Universal Robots PolyScope program: wrs2020_taskboard_pulley.urp

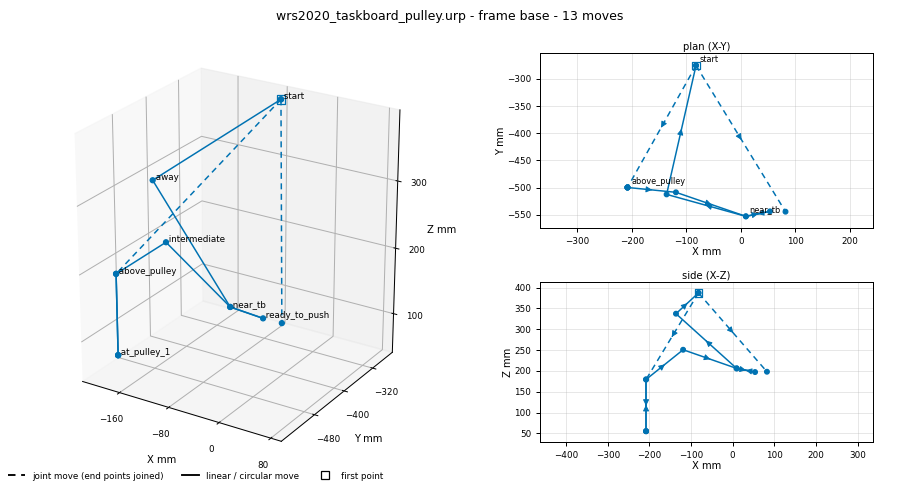
[picture p0: tool path of wrs2020_taskboard_pulley.urp in frame base, 13 of 13 moves have a stored position in this frame; points joined in program order, loops and branches not executed]
Program wrs2020_taskboard_pulley (installation=default directory=/programs/usbdisk createdIn=5.6.0.90886 lastSavedIn=5.6.0.90886 robotSerialNumber=20205500180)
Calibrated DH parameters: a=[0.000135, -0.030981, -0.334292, 0.000083, 0.000088, 0]; d=[0.162656, 258.79096, -331.603246, 72.945842, 0.099724, 0.099562]; alpha=[1.569535, 0.001639, 0.002824, 1.569633, -1.569323, 0]; deltaTheta=[0, 1.497881, -2.049261, 0.551379, 0, 0]
Robot Program (runOnlyOnce=true)
  MoveJ speed 60 deg/s, acceleration 80 deg/s^2 (useActiveTCP=false) tcp=gripper_140_tip; feature=Base
    Waypoint start: TCP in base x=-82.102 y=-275.549 z=387.348 mm, rx=-0.1814 ry=-3.1114 rz=0.2863 rad; joints [35.849, -127.007, 98.51, -68.6, -82.206, -47.132] deg; TCP offset x=0 y=0 z=220 mm, rx=0 ry=0 rz=0 rad
  URCap Gripper (Robotiq_Grippers, Robotiq Inc.) dataModel(position=44.705882352941174, force=100.0, speed=100.0, positionInDouble=44.705882352941174, forceInDouble=100.0, speedInDouble=100.0, slaveIds=[9], blocking=true)
  MoveJ speed 120 deg/s, acceleration 80 deg/s^2 (useActiveTCP=false) tcp=gripper_140_tip; feature=Base
    Waypoint above_pulley: TCP in base x=-208.011 y=-499.592 z=179.536 mm, rx=2.2188 ry=-2.2117 rz=-0.0634 rad; joints [54.601, -83.96, 96.653, -102.683, -92.188, -125.564] deg
  MoveL speed 250 mm/s, acceleration 1200 mm/s^2 (useActiveTCP=false) tcp=gripper_140_tip; feature=Base
    Waypoint at_pulley_1: motionParameters(jointSpeed=1.047198 jointAcceleration=1.396263 cartesianSpeed=0.5 cartesianAcceleration=1.2); TCP in base x=-208.011 y=-499.592 z=55.279 mm, rx=2.2188 ry=-2.2117 rz=-0.0634 rad; joints [54.587, -77.543, 108.66, -121.106, -92.18, -125.517] deg
  URCap Gripper (Robotiq_Grippers, Robotiq Inc.) dataModel(position=100.0, force=0.0, speed=0.0, positionInDouble=100.0, forceInDouble=0.0, speedInDouble=0.0, slaveIds=[9], blocking=true)
  URCap Gripper (Robotiq_Grippers, Robotiq Inc.) dataModel(position=56.86274509803921, force=0.0, speed=0.0, positionInDouble=56.86274509803921, forceInDouble=0.0, speedInDouble=0.0, slaveIds=[9], blocking=true)
  MoveL speed 500 mm/s, acceleration 1200 mm/s^2 (useActiveTCP=false) tcp=gripper_140_tip; feature=Base
    Waypoint at_pulley_2: motionParameters(jointSpeed=1.047198 jointAcceleration=1.396263 cartesianSpeed=0.5 cartesianAcceleration=1.2); TCP in base x=-207.996 y=-499.585 z=55.27 mm, rx=-0.009 ry=-3.1069 rz=-0.0353 rad; joints [54.588, -77.543, 108.661, -121.105, -92.181, -35] deg
  URCap Gripper (Robotiq_Grippers, Robotiq Inc.) dataModel(position=100.0, force=0.0, speed=0.0, positionInDouble=100.0, forceInDouble=0.0, speedInDouble=0.0, slaveIds=[9], blocking=true)
  URCap Gripper (Robotiq_Grippers, Robotiq Inc.) dataModel(position=56.86274509803921, force=0.0, speed=0.0, positionInDouble=56.86274509803921, forceInDouble=0.0, speedInDouble=0.0, slaveIds=[9], blocking=true)
  MoveL speed 500 mm/s, acceleration 1200 mm/s^2 (useActiveTCP=false) tcp=gripper_140_tip; feature=Base
    Waypoint at_pulley_1: motionParameters(jointSpeed=1.047198 jointAcceleration=1.396263 cartesianSpeed=0.5 cartesianAcceleration=1.2); TCP in base x=-208.011 y=-499.592 z=55.279 mm, rx=2.2188 ry=-2.2117 rz=-0.0634 rad; joints [54.587, -77.543, 108.66, -121.106, -92.18, -125.517] deg
  URCap Gripper (Robotiq_Grippers, Robotiq Inc.) dataModel(position=100.0, force=0.0, speed=0.0, positionInDouble=100.0, forceInDouble=0.0, speedInDouble=0.0, slaveIds=[9], blocking=true)
  MoveL speed 250 mm/s, acceleration 250 mm/s^2 (useActiveTCP=false) tcp=gripper_140_tip; feature=Base
    Waypoint above_pulley: TCP in base x=-208.011 y=-499.592 z=179.536 mm, rx=2.2188 ry=-2.2117 rz=-0.0634 rad; joints [54.601, -83.96, 96.653, -102.683, -92.188, -125.564] deg
    Waypoint intermediate: motionParameters(blendRadius=0.05); TCP in base x=-119.041 y=-508.485 z=250.905 mm, rx=-1.87 ry=2.1339 rz=-0.5992 rad; joints [46.177, -86.722, 91.166, -81.687, -65.2, -129.14] deg
  MoveL speed 250 mm/s, acceleration 250 mm/s^2 (useActiveTCP=false) tcp=gripper_140_tip; feature=Base
    Waypoint near_tb: TCP in base x=9.516 y=-552.663 z=206.118 mm, rx=-1.2151 ry=1.2878 rz=-1.2829 rad; joints [46.82, -54.652, 84.012, -32.299, -37.921, -179.667] deg
    Waypoint ready_to_push: TCP in base x=53.765 y=-543.482 z=197.335 mm, rx=-1.1908 ry=1.1936 rz=-1.2641 rad; joints [50.694, -52.534, 85.468, -29.603, -37.71, -184.158] deg
  Force Frame feature=Joint_6_name; selection=[1, 1, 1, 0, 0, 0]; wrench=[0, 0, 10, 0, 0, 0]; limitsForce=[0.15, 0.15, 0.01, 1.047198, 1.047198, 1.047198]; limitsMotion=[0.1, 0.1, 0.1, 0.349066, 0.349066, 0.349066]
    Wait Sleep waitTime=3
    Loop Counting (count=5) loopVariable(name=Loop_1)
      SuppressedNode
        MoveL speed 5 mm/s, acceleration 1200 mm/s^2 (useActiveTCP=true) feature=Base
          MoveDirectionNode (selectedDirection=XPlus toolParams=0.005, 1.2) feature=Joint_6_name
            Until DISTANCE (allowActions=false deceleration=3 distanceNodeType=STOP) Distance=0.002; motionParameters(blendRadius=0)
          MoveDirectionNode (selectedDirection=XMinus toolParams=0.005, 1.2) feature=Joint_6_name
            Until DISTANCE (allowActions=false deceleration=3 distanceNodeType=STOP) Distance=0.002; motionParameters(blendRadius=0)
          MoveDirectionNode (selectedDirection=XMinus toolParams=0.005, 1.2) feature=Joint_6_name
            Until DISTANCE (allowActions=false deceleration=3 distanceNodeType=STOP) Distance=0.002; motionParameters(blendRadius=0)
          MoveDirectionNode (selectedDirection=XPlus toolParams=0.005, 1.2) feature=Joint_6_name
            Until DISTANCE (allowActions=false deceleration=3 distanceNodeType=STOP) Distance=0.002; motionParameters(blendRadius=0)
          MoveDirectionNode (selectedDirection=YPlus toolParams=0.005, 1.2) feature=Joint_6_name
            Until DISTANCE (allowActions=false deceleration=3 distanceNodeType=STOP) Distance=0.002; motionParameters(blendRadius=0)
          MoveDirectionNode (selectedDirection=YMinus toolParams=0.005, 1.2) feature=Joint_6_name
            Until DISTANCE (allowActions=false deceleration=3 distanceNodeType=STOP) Distance=0.002; motionParameters(blendRadius=0)
          MoveDirectionNode (selectedDirection=YMinus toolParams=0.005, 1.2) feature=Joint_6_name
            Until DISTANCE (allowActions=false deceleration=3 distanceNodeType=STOP) Distance=0.002; motionParameters(blendRadius=0)
          MoveDirectionNode (selectedDirection=YPlus toolParams=0.005, 1.2) feature=Joint_6_name
            Until DISTANCE (allowActions=false deceleration=3 distanceNodeType=STOP) Distance=0.002; motionParameters(blendRadius=0)
      Loop Counting (count=6) loopVariable(name=Loop_2)
        MoveL speed 5 mm/s, acceleration 1200 mm/s^2 (useActiveTCP=false) tcp=gripper_140_tip; feature=Base
          MoveDirectionNode (toolParams=0.005, 1.2) expression=[sin((Loop_2-1)/6),cos((Loop_2-1)/6),0.0]; feature=Joint_6_name
            Until DISTANCE (allowActions=false deceleration=3 distanceNodeType=STOP) Distance=0.003; motionParameters(blendRadius=0)
        SuppressedNode
          dist := pose_dist(fully_pushed, Joint_6_name)
        SuppressedNode
          Popup Message (haltProgram=false inputType=Variable) variable=dist
        Wait Sleep waitTime=0.5
  Popup Message (haltProgram=false message=done, will open inputType=Text)
  URCap Gripper (Robotiq_Grippers, Robotiq Inc.) dataModel(position=41.96078431372549, force=100.0, speed=100.0, positionInDouble=41.96078431372549, forceInDouble=100.0, speedInDouble=100.0, slaveIds=[9], blocking=true)
  MoveL speed 250 mm/s, acceleration 1200 mm/s^2 (useActiveTCP=true) feature=Base
    MoveDirectionNode (selectedDirection=ZMinus toolParams=0.25, 1.2) feature=Joint_6_name
      Until DISTANCE (allowActions=false deceleration=3 distanceNodeType=STOP) Distance=0.015; motionParameters(blendRadius=0)
  URCap Gripper (Robotiq_Grippers, Robotiq Inc.) dataModel(position=75.68627450980392, force=100.0, speed=100.0, positionInDouble=75.68627450980392, forceInDouble=100.0, speedInDouble=100.0, slaveIds=[9], blocking=true)
  MoveL speed 250 mm/s, acceleration 1200 mm/s^2 (useActiveTCP=true) feature=Base
    MoveDirectionNode (selectedDirection=ZPlus) feature=Joint_6_name
      Until TOOL_CONTACT_DETECTION (allowActions=false retraction=0.04 decelerationAcceleration=3 decelerationAngularAcceleration=34.906585)
  MoveL speed 250 mm/s, acceleration 1200 mm/s^2 (useActiveTCP=false) tcp=gripper_140_tip; feature=Base
    Waypoint near_tb: TCP in base x=9.516 y=-552.663 z=206.118 mm, rx=-1.2151 ry=1.2878 rz=-1.2829 rad; joints [46.82, -54.652, 84.012, -32.299, -37.921, -179.667] deg
    Waypoint away: motionParameters(blendRadius=0.05); TCP in base x=-136.161 y=-512.303 z=337.477 mm, rx=2.1588 ry=-1.5967 rz=1.3013 rad; joints [29.498, -97.585, 100.743, -75.77, -39.512, -175.862] deg
    Waypoint start: TCP in base x=-82.102 y=-275.549 z=387.348 mm, rx=-0.1814 ry=-3.1114 rz=0.2863 rad; joints [35.849, -127.007, 98.51, -68.6, -82.206, -47.132] deg
  Halt
  MoveJ speed 60 deg/s, acceleration 80 deg/s^2 (useActiveTCP=true) feature=Base
    Waypoint fully_pushed: TCP in base x=82.304 y=-544.056 z=198.103 mm, rx=-1.1908 ry=1.1938 rz=-1.2643 rad; joints [52.959, -53.905, 87.77, -30.349, -35.433, -184.386] deg
